PROGRAM MAIN
VAR
    iCount : INT;
END_VAR

iCount:=iCount+1;

END_PROGRAM

(* stored: Version 1.1.0.1, ProductVersion 3.1.4024.12
   POU MAIN: Id {790d3e76-e969-4252-8a13-08f65b5816ff}, SpecialFunc None *)
